# EPICS autosave request: iocs/andorIOC/iocBoot/iocAndor/auto_settings.req
file "ADBase_settings.req",       P=$(P),  R=cam1:
file "andorCCD_settings.req",     P=$(P),  R=cam1:
file "shamrock_settings.req",     P=$(P),  R=sham1:
file "NDFile_settings.req",       P=$(P),  R=cam1:
file "NDPluginBase_settings.req", P=$(P),  R=image1:
file "NDStdArrays_settings.req",  P=$(P),  R=image1:
file "commonPlugin_settings.req", P=$(P)
